# B&R Automation Studio project PLC
Automation Studio 4.9

## Configuration Config1

CPU X20CP0484, AutomationRuntime H4.90, Build 4.1.2, Safety 0.0, Vc 

### Task classes (Cpu.sw)
```
Cyclic#1 (cycle 10000 us, tolerance 10000 us):
  PullUpdate <- PullUpdate.prg
Binaries: FWRules, udbdef, arsvcreg, TCData, User, arconfig, Role, iomap, asfw, ashwac, ashwd, sysconf, backupConf
Libraries: MpBackup, MpBase, FileIO, runtime, asarcfg, sys_lib, astime, asieccon, brsystem, ArProject, standard
```

### Hardware
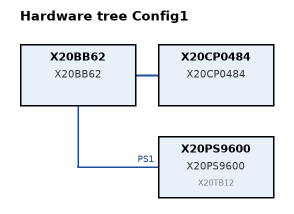
```
X20BB62 : X20BB62 v1.3.0.0
X20CP0484 : X20CP0484 v1.8.1.0  [SL -> X20BB62.SL1]
  Connector IF2:
    ActivateDevice = 1
    ActivateSnmp = 2
  ConfigurationID = HorribleSoftware
  ConfigVersion = 1.2.3
  UserPartitionSize = 100
  EnableUsbRemoteInstall = 1
  EnableCfRemoteInstall = 1
  TimerDeviceType = SWIOTIMER
  Cyclic1Duration = 10000
  Cyclic1Tolerance = 10000
  Cyclic2Duration = 20000
  Cyclic2Tolerance = 20000
  Cyclic3Duration = 50000
  Cyclic3Tolerance = 50000
  Cyclic4Duration = 100000
  Cyclic4Tolerance = 100000
  Cyclic5Duration = 200000
  Cyclic5Tolerance = 200000
  Cyclic6Duration = 500000
  Cyclic6Tolerance = 500000
  Cyclic7Duration = 1000000
  Cyclic7Tolerance = 1000000
  Cyclic8Duration = 10000
  Cyclic8Tolerance = 30000000
  FileDevice1
  FileDeviceName1 = USER
  FileDevicePath1 = USER_PATH
  FileDevice2
  FileDeviceName2 = ROOT
  FileDevicePath2 = F:/
  FtpUser1
  FtpUsername1 = admin
  FtpUserPassword1 = aJYGXaJ9VUePXTlsiEuc8Wdng+6l4gdEbbX02y4mLPg=
  FtpUserSalt1 = arZaZjbb
  FTPAccessRight1 = 0
  FtpUser2
  FtpUsername2 = superuser
  FtpUserPassword2 = RfTOMjpK21SCeBQ66ZoRWWPmgaIpiJPQiIUJFzVOu94=
  FtpUserSalt2 = 9qhK3iVE
  FTPAccessRight2 = 0
  FTPdevice2 = ALL
  ActivateOpcUa = 1
  OpcUaInformationModels_PV_Version = 1
X20PS9600 : X20PS9600 v1.6.1.0  [PS -> X20BB62.PS1; SS1 -> X20TB12.SS]
X20TB12 : X20TB12 v1.0.0.0
```

## Logical view

Binary libraries used (declarations not repeated): operator, runtime, astime, AsIecCon, MpBackup 5.24.3, MpBase, FileIO, ArProject, standard


### Program Logical/PullUpdate (IEC)

#### Variables.var
```iecst
VAR
	state : USINT;
	DevLink_0 : DevLink;
	DirCopy_0 : DirCopy;
	updateFolderName : STRING[80];
	reset : BOOL;
	ArProjectGetInfo_0 : ArProjectGetInfo;
	DownloadUpdate : BOOL;
	ExecuteUpdate : BOOL;
	ArProjectInstallPackage_0 : ArProjectInstallPackage;
	CheckVersion : BOOL;
	ArProjectGetPackageInfo_0 : ArProjectGetPackageInfo;
END_VAR
```

#### Main.st
```iecst
PROGRAM _INIT

	// Read current version
	WHILE NOT ArProjectGetInfo_0.Done AND NOT ArProjectGetInfo_0.Error DO
		ArProjectGetInfo_0.Execute := TRUE;
		ArProjectGetInfo_0();
	END_WHILE
	// See Current Version in: ArProjectGetInfo_0.ConfigurationVersion & ArProjectGetInfo_0.ConfigurationID

END_PROGRAM

PROGRAM _CYCLIC

	CASE state OF

		0:
			DevLink_0.enable := TRUE;
			DevLink_0.pDevice := ADR('PLCUPDATE');
			DevLink_0.pParam := ADR('/SIP=192.168.30.64 /PROTOCOL=ftp /USER=update /PASSWORD=update');
			DevLink_0();

			IF DevLink_0.status = ERR_OK OR DevLink_0.status = fiERR_DEVICE_ALREADY_EXIST THEN
				DevLink_0.enable := FALSE;
				DevLink_0();
				state := 10;
			ELSIF DevLink_0.status <> ERR_FUB_BUSY THEN
				state := 222;
			END_IF

		10:
			IF DownloadUpdate THEN
				// Will download update with name 'updateFolderName'
				DownloadUpdate := FALSE;
				state := 20;
			ELSIF CheckVersion THEN
				// Will check version of update with name 'updateFolderName'
				CheckVersion := FALSE;
				ArProjectGetPackageInfo_0.Execute := FALSE;
				ArProjectGetPackageInfo_0();
				state := 30;
			ELSIF ExecuteUpdate THEN
				// Will Execute update with name 'updateFolderName'
				ExecuteUpdate := FALSE;
				ArProjectInstallPackage_0.Execute := FALSE;
				ArProjectInstallPackage_0();
				state := 40;
			END_IF

		20:
			DirCopy_0.enable := TRUE;
			DirCopy_0.pSrcDev := ADR('PLCUPDATE');
			DirCopy_0.pSrcDir := ADR(updateFolderName);
			DirCopy_0.pDestDev := ADR('ROOT');
			DirCopy_0.option := fiOVERWRITE;
			DirCopy_0();

			IF DirCopy_0.status = ERR_OK THEN
				DirCopy_0.enable := FALSE;
				DirCopy_0();
				state := 10;
			ELSIF DirCopy_0.status <> ERR_FUB_BUSY THEN
				state := 222;
			END_IF

		30:
			ArProjectGetPackageInfo_0.Execute := TRUE;
			ArProjectGetPackageInfo_0.DeviceName := 'ROOT';
			ArProjectGetPackageInfo_0.FilePath := CONCAT(updateFolderName,'/Default_X20CP04xx/pipconfig.xml');
			ArProjectGetPackageInfo_0();

			IF ArProjectGetPackageInfo_0.Done THEN
				state := 10;
			ELSIF ArProjectGetPackageInfo_0.Error THEN
				state := 222;
			END_IF

		40:
			ArProjectInstallPackage_0.Execute := TRUE;
			ArProjectInstallPackage_0.DeviceName := 'ROOT';
			ArProjectInstallPackage_0.FilePath := CONCAT(updateFolderName,'/Default_X20CP04xx/pipconfig.xml');
			ArProjectInstallPackage_0();

			IF ArProjectInstallPackage_0.Done THEN
				state := 10;
			ELSIF ArProjectInstallPackage_0.Error THEN
				state := 222;
			END_IF

		222:

			IF reset THEN
				reset := FALSE;
				DirCopy_0.enable := FALSE;
				DirCopy_0();
				DevLink_0.enable := FALSE;
				DevLink_0();
				ArProjectGetPackageInfo_0.Execute := FALSE;
				ArProjectGetPackageInfo_0();
				ArProjectInstallPackage_0.Execute := FALSE;
				ArProjectInstallPackage_0();
				state := 0;
			END_IF

	END_CASE

END_PROGRAM

PROGRAM _EXIT

END_PROGRAM
```

Listed in the project but not available here: Logical/Global.typ, Logical/Global.var
